VAR_GLOBAL
	itf_content : ST_adsITF;
END_VAR

(* stored: Version 1.1.0.1, ProductVersion 3.1.4024.11
   GVL GVL_adsITF: Id {9535baf7-3d8c-4f3b-ab24-c8dbbcff5b72} *)
